// TIA Portal V20 export
FUNCTION_BLOCK "Simulation_Interface"   // FB106, LAD
// stored: Access Published, MemoryReserve 100, SetENOAutomatically false
   VAR_INPUT
      jrDetectUnused : Bool;
      I2S : "LER_typeInspectionToStack";
   END_VAR
   VAR_OUTPUT
      S2I : "LER_typeStackToInspection";
   END_VAR
   VAR
      instTON { S7_SetPoint := 'True'} : Array[0..9] of TON_TIME;
   END_VAR
   VAR_TEMP
      tempData : "LER_typeCommonData";   // TCP/IP STK data
   END_VAR
   VAR CONSTANT
      delayTime : Time := T#1s;
   END_VAR
BEGIN

REGION Network 1
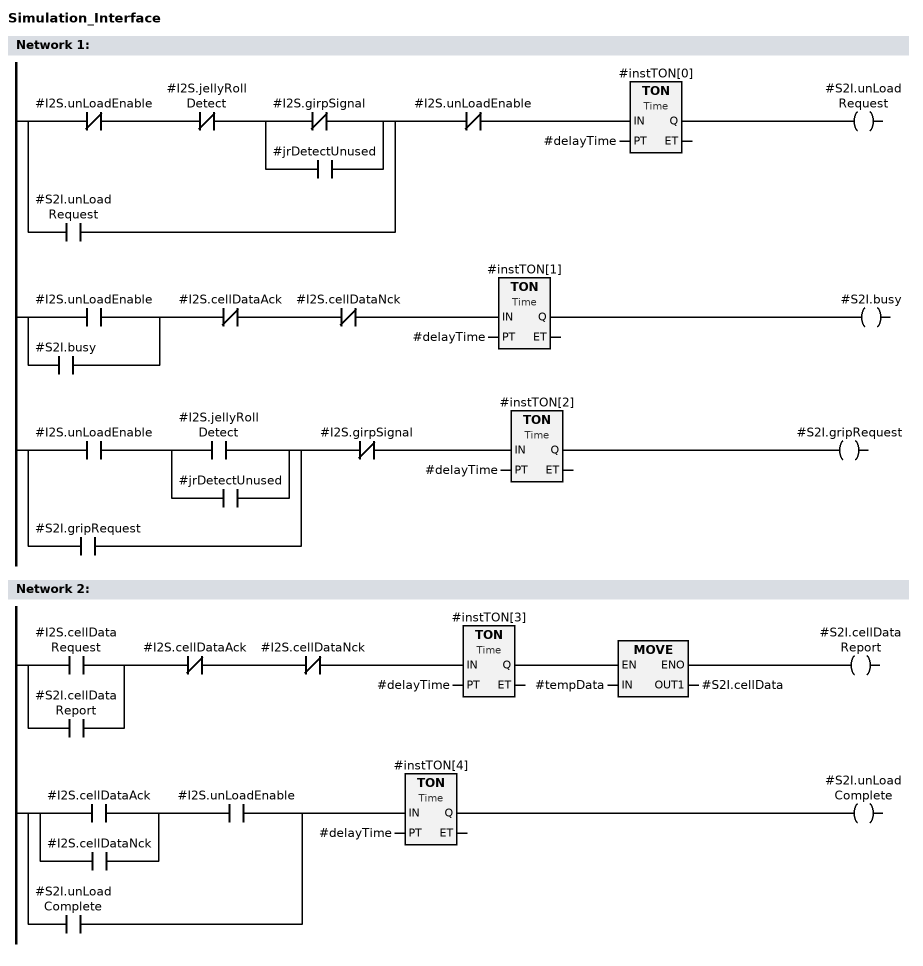
   RUNG wire#powerrail
      I_Contact( #I2S.unLoadEnable )
      I_Contact( #I2S.jellyRollDetect )
      wire#w1
      I_Contact( #I2S.girpSignal )
      wire#w2
      I_Contact( #I2S.unLoadEnable )
      { S7_Templates := "time_type := Time" } #instTON[0].TON(pt := #delayTime, et =>)
      Coil( #S2I.unLoadRequest )
   END_RUNG
   RUNG wire#w1
      Contact( #jrDetectUnused )
   END_RUNG wire#w2
   RUNG wire#powerrail
      Contact( #S2I.unLoadRequest )
   END_RUNG wire#w2
   RUNG wire#powerrail
      Contact( #I2S.unLoadEnable )
      wire#w3
      I_Contact( #I2S.cellDataAck )
      I_Contact( #I2S.cellDataNck )
      { S7_Templates := "time_type := Time" } #instTON[1].TON(pt := #delayTime, et =>)
      Coil( #S2I.busy )
   END_RUNG
   RUNG wire#powerrail
      Contact( #S2I.busy )
   END_RUNG wire#w3
   RUNG wire#powerrail
      Contact( #I2S.unLoadEnable )
      wire#w4
      Contact( #I2S.jellyRollDetect )
      wire#w5
      I_Contact( #I2S.girpSignal )
      { S7_Templates := "time_type := Time" } #instTON[2].TON(pt := #delayTime, et =>)
      Coil( #S2I.gripRequest )
   END_RUNG
   RUNG wire#w4
      Contact( #jrDetectUnused )
   END_RUNG wire#w5
   RUNG wire#powerrail
      Contact( #S2I.gripRequest )
   END_RUNG wire#w5
   // the same network as SCL:
   #instTON[0].TON(IN := ((NOT #I2S.unLoadEnable AND NOT #I2S.jellyRollDetect AND (NOT #I2S.girpSignal OR #jrDetectUnused)) OR #S2I.unLoadRequest) AND NOT #I2S.unLoadEnable,
                   PT := #delayTime);
   #S2I.unLoadRequest := #instTON[0].Q;
   #instTON[1].TON(IN := (#I2S.unLoadEnable OR #S2I.busy) AND NOT #I2S.cellDataAck AND NOT #I2S.cellDataNck,
                   PT := #delayTime);
   #S2I.busy := #instTON[1].Q;
   #instTON[2].TON(IN := ((#I2S.unLoadEnable AND (#I2S.jellyRollDetect OR #jrDetectUnused)) OR #S2I.gripRequest) AND NOT #I2S.girpSignal,
                   PT := #delayTime);
   #S2I.gripRequest := #instTON[2].Q;
END_REGION

REGION Network 2
   RUNG wire#powerrail
      Contact( #I2S.cellDataRequest )
      wire#w1
      I_Contact( #I2S.cellDataAck )
      I_Contact( #I2S.cellDataNck )
      { S7_Templates := "time_type := Time" } #instTON[3].TON(pt := #delayTime, et =>)
      Move(in := #tempData, out1 => #S2I.cellData)
      Coil( #S2I.cellDataReport )
   END_RUNG
   RUNG wire#powerrail
      Contact( #S2I.cellDataReport )
   END_RUNG wire#w1
   RUNG wire#powerrail
      Contact( #I2S.cellDataAck )
      wire#w2
      Contact( #I2S.unLoadEnable )
      wire#w3
      { S7_Templates := "time_type := Time" } #instTON[4].TON(pt := #delayTime, et =>)
      Coil( #S2I.unLoadComplete )
   END_RUNG
   RUNG wire#powerrail
      Contact( #I2S.cellDataNck )
   END_RUNG wire#w2
   RUNG wire#powerrail
      Contact( #S2I.unLoadComplete )
   END_RUNG wire#w3
   // the same network as SCL:
   #instTON[3].TON(IN := (#I2S.cellDataRequest OR #S2I.cellDataReport) AND NOT #I2S.cellDataAck AND NOT #I2S.cellDataNck,
                   PT := #delayTime);
   IF #instTON[3].Q THEN #S2I.cellData := #tempData; END_IF;
   #S2I.cellDataReport := #instTON[3].Q;
   #instTON[4].TON(IN := ((#I2S.cellDataAck OR #I2S.cellDataNck) AND #I2S.unLoadEnable) OR #S2I.unLoadComplete,
                   PT := #delayTime);
   #S2I.unLoadComplete := #instTON[4].Q;
END_REGION
END_FUNCTION_BLOCK
